Staubli VAL3: deletListItem.pgx

public program deletListItem(string& x_sList[], num x_nFirst, num& x_nSelect, bool& x_bListRefresh, bool& x_bRes)
  local string l_sYesNo[2]
  local num l_i
begin
  //F3:
  //x_nFirst:>=n(n>=1),按顺序保留的前n项
  //x_nFirst:0 不按顺序保留最后一项
  //x_nFirst:-1 全部删除,x_sList[0]=""
  x_bListRefresh=false
  x_bRes=false
  l_sYesNo[0]="是"
  l_sYesNo[1]="否"
  call user:questionDialog("是否删除该项?",l_sYesNo,l_i)
  if l_i==0 or l_i==1
    //
    x_nFirst=roundDown(x_nFirst)
    if x_nFirst==0
      if size(x_sList)==1
        popUpMsg("不能删除项!")
        return
      endIf
    endIf
    if size(x_sList)<=x_nFirst or x_nSelect<x_nFirst
      popUpMsg("不能删除项!")
      return
    endIf
    if size(x_sList)==1 and x_nFirst==-1
      x_sList=""
      x_bRes=true
      x_bListRefresh=true
      return
    endIf
    delete(x_sList[x_nSelect])
    x_nSelect=x_nSelect-1
    if x_nSelect<0
      x_nSelect=0
    endIf
    x_bListRefresh=true
    x_bRes=true
  endIf
end
